(* CoDeSys 2.3.9.47 project: ATS_P3.pro *)
(* Libraries: STANDARD.LIB 5.6.98 12:03:02 *)

(* Task configuration *)
TASK Standard (PRIORITY := 0, INTERVAL := T#10ms);
	MAIN
END_TASK

(* Global variable list: Global_Variables *)
VAR_GLOBAL
	b_global_calc_correct : BOOL := FALSE;
END_VAR

(* POU MAIN, ST *)
PROGRAM MAIN
VAR
(*OPERANDS*)	
	r_op_1	: REAL	:= 5;
	r_op_2	: REAL	:= 3;
(*RESULTS*)
	r_sum	: REAL	;
	r_dif	: REAL	;
	r_pro	: REAL	;
	r_quo	: REAL	;
END_VAR
(*Addition*)
r_sum := AdditionFunction(r_op_1, r_op_2);
(*Subtraction*)
r_dif := SubtractionFunction(r_op_1, r_op_2);
(*Multiplication*)
r_pro := MultiplicationFunction(r_op_1, r_op_2);
(*Division*)
r_quo := DivisionFunction(r_op_1, r_op_2);

DoSomeMath;
res := DoSomeMath
END_PROGRAM

(* POU AdditionFunction, ST *)
FUNCTION AdditionFunction : REAL
VAR_INPUT
	r_operand_1 : REAL;
	r_operand_2 : REAL;
END_VAR
VAR
	r_result	: REAL;
END_VAR
(* CALCULATE SUM OF TWO REAL's *)
AdditionFunction := (r_operand_1 + r_operand_2);
END_FUNCTION

(* POU SubtractionFunction, ST *)
FUNCTION SubtractionFunction : REAL
VAR_INPUT
	r_operand_1	:	REAL;
	r_operand_2	:	REAL;
END_VAR
VAR
	r_result	:	REAL;
END_VAR
(* CALCULATE DIFFERENCE BETWEEN TWO REAL's *)
SubtractionFunction := (r_operand_1 - r_operand_2);
END_FUNCTION

(* POU MultiplicationFunction, ST *)
FUNCTION MultiplicationFunction : REAL
VAR_INPUT
	r_operand_1	:	REAL;
	r_operand_2	:	REAL;
END_VAR
VAR
	r_result	:	REAL;
END_VAR
(* CALCULATE PRODUCT OF TWO REAL's *)
MultiplicationFunction := r_operand_1 * r_operand_2;
END_FUNCTION

(* POU DivisionFunction, ST *)
FUNCTION DivisionFunction : REAL
VAR_INPUT
	r_operand_1 : REAL;
	r_operand_2	: REAL;
END_VAR
VAR
	r_result	: REAL;
END_VAR
(* CALCULATE QUOTIENT OF TWO REAL's *)
IF r_operand_2 = 0 THEN
	DivisionFunction := 0;
ELSE
	DivisionFunction := r_operand_1/r_operand_2;
END_IF
END_FUNCTION

(* POU DoSomeMath, ST *)
PROGRAM DoSomeMath
VAR
(*OPERANDS*)	
	r_op_1	: REAL	;
	r_op_2	: REAL	;
(*RESULTS*)
	r_res	: REAL	;
END_VAR
(*Addition*)
r_sum := AdditionFunction(r_op_1, r_op_2);
(*Subtraction*)
r_dif := SubtractionFunction(r_op_1, r_op_2);
(*Multiplication*)
r_pro := MultiplicationFunction(r_op_1, r_op_2);
(*Division*)
r_quo := DivisionFunction(r_op_1, r_op_2);
END_PROGRAM
